Staubli VAL3: PlasticMain.pjx

--- PlasticMain.pjx ---
Parameters version=s7.0 stackSize=400000 millimeterUnit=true
Program file=__ts_english.pgx
Program file=__ts_german.pgx
Program file=__ts_swedish.pgx
Program file=_globals.pgx
Program file=changeLog.pgx
Program file=checkRobotPos.pgx
Program file=checkTaskStates.pgx
Program file=cleanUpDataBase.pgx
Program file=controlTasks.pgx
Program file=createLicense.pgx
Program file=detailedStack.pgx
Program file=loadApplication.pgx
Program file=loadLibraries.pgx
Program file=loadSysData.pgx
Program file=loadUserProgram.pgx
Program file=loadVersionInfo.pgx
Program file=logo.pgx
Program file=parseStackInfo.pgx
Program file=processEvents.pgx
Program file=run.pgx
Program file=saveApplication.pgx
Program file=start.pgx
Program file=startUpTask.pgx
Program file=status.pgx
Program file=stop.pgx
Program file=taskKill.pgx
Program file=taskKiller.pgx
Data file=PlasticMain.dtx
Library alias=rob path=Disk://Plastic/Prototypes/modRobot/modRobot.pjx autoload=false
Library alias=data path=Disk://Plastic/templates/sysDataTemplate/sysDataTemplate.pjx autoload=false
Library alias=secu path=Disk://Plastic/Prototypes/modSafety/modSafety.pjx autoload=false
Library alias=util path=Disk://Plastic/Prototypes/modBackup/modBackup.pjx autoload=false
Library alias=FUN path=Disk://Plastic/templates/tempSysFuncCall/tempSysFuncCall.pjx autoload=false
Library alias=fun path=Disk://Plastic/Prototypes/modFunction/modFunction.pjx autoload=false
Library alias=ui path=Disk://Plastic/Prototypes/modUserDisp/modUserDisp.pjx autoload=false
Library alias=prg path=Disk://Plastic/templates/tempUserProgram/tempUserProgram.pjx autoload=false
Library alias=USER path=Disk://Plastic/templates/tempIoUser/tempIoUser.pjx autoload=false
Library alias=app path=Disk://Plastic/templates/tempApplication/tempApplication.pjx
Library alias=appTmp path=Disk://Plastic/templates/tempApplication/tempApplication.pjx
Library alias=evt path=Disk://Plastic/Prototypes/modEvents/modEvents.pjx autoload=false
Library alias=SYS path=Disk://io_System/io_System.pjx
Library alias=str path=Disk://Libraries/stringHandling/stringHandling.pjx
Library alias=list path=Disk://Libraries/listHandling/listHandling.pjx
Library alias=upd path=Disk://Plastic/Prototypes/modUpdater/modUpdater.pjx autoload=false
Library alias=stat path=Disk://Plastic/Prototypes/modStatus/modStatus.pjx autoload=false
Library alias=lang path=Disk://Plastic/i18n/i18n.pjx
Library alias=db path=Disk://Plastic/Prototypes/modDatabase/modDatabase.pjx autoload=false
Library alias=usr path=Disk://Plastic/Prototypes/modUserIO/modUserIO.pjx autoload=false
Library alias=hw path=Disk://Libraries/hardware/hardware.pjx
Library alias=msl path=Disk://Plastic/Prototypes/modMsl/modMsl.pjx autoload=false
Library alias=customModule path=Disk://Plastic/Prototypes/modCustom/modCustom.pjx autoload=false
Library alias=userIO path=Disk://zUserIODef/zUserIODef.pjx autoload=false
Library alias=monitor path=Disk://Plastic/Prototypes/modMonitor/modMonitor.pjx autoload=false
Library alias=debug path=Disk://Libraries/debug/debug.pjx

--- PlasticMain.dtx ---
num nPLCRestartCnt
string programList
string sTaskName[3]
  [0] = "PLC_Main"
  [1] = "MP_MainPRG"
  [2] = "SR_HomeReturn"
string sVersion
string sBuildNumber
bool bFirstLoad = true
bool bStartUp
bool homeFlag
bool overrun
string sRawList
string sCopyRight = "Plastics (C) 2006-2011 V"

--- __ts_german.pgx ---
program __ts_german()
begin
  //
end

--- __ts_swedish.pgx ---
program __ts_swedish()
begin
  //
end

--- _globals.pgx ---
program _globals()
begin
    //\brief
  //
  //\version
  //4.3c
  //
//!version 4.3c
end

--- controlTasks.pgx ---
program controlTasks()
  local bool bResult
  local num nResult
begin
    //
  //\var bResult
  //\var nResult
  //
//=========================================================================
  // START PLC
  //=========================================================================
  if (taskStatus(sTaskName[0])==-1)
    taskCreate (sTaskName[0]),10,app:PLC_MainPLC()
  endIf
  // if PLC task is stopped due to an runtime error it should be restarted immediately
  if (taskStatus(sTaskName[0])>1) and nPLCRestartCnt<5
    if nPLCRestartCnt<5
      call ui:error("PLC task "+sTaskName[0]+" of "+data:sApplication+" died unexpectedly with error #"+toString(".0",taskStatus(sTaskName[0])))
      nPLCRestartCnt=nPLCRestartCnt+1
      nResult=1
    else
      call ui:question("PLC task "+sTaskName[0]+" died to often! Do you want to continue?",nResult)
      if nResult==1
        nPLCRestartCnt=0
      endIf
    endIf
    if nResult==1
      taskKill(sTaskName[0])
      delay(1)
      taskCreate (sTaskName[0]),10,app:PLC_MainPLC()
    endIf
  endIf
  //!change: 11.03.08, vdg: try to restart PLC task when robot leaves home position
  if !SYS:bRobotHome and homeFlag and nPLCRestartCnt>=5
    nPLCRestartCnt=0
  endIf
  homeFlag=SYS:bRobotHome
  //=========================================================================
  // START PRODUCTION CYCLE
  //=========================================================================
  if SYS:bStartProdCycle and SYS:bRobotHome and (taskStatus(sTaskName[1])==-1)
    SYS:bStartProdCycle=false
    call taskKill(sTaskName[2],bResult)
    if !bResult
      // killing the task failed, because it is being debugged?!
      call ui:popUp((("Cycle start not possible!/nPlease check if task HR_HomeReturn exists in task manager!")),0,false)
    else
      // inform operator that force recording is active
      if SYS:bRecordForce
        call ui:popUp((("Recording is active!/nDeactivate it in Advanced Settings->Test Run->Edit System Settings")),data:nMsgTimeOut,false)
      endIf
      resetMotion()
      restartMove()
      // reduce monitor speed to data:nSpeedAfterLoad if this is the first start cycle
      if SYS:bFirstRunAfterL
        ///TODO
        //$setSpeed(min(data:nSpeedAfterLoad,speedScale()))
        call fun:setSpeed(min(data:nSpeedAfterLoad,getMonitorSpeed()))
        // give the system some time to adjust the monitor speed before
        // MP_MainProgram is actually started
        delay(0.4)
        SYS:bFirstRunAfterL=false
        //
        //!change 18.05.06, vdg: activate test run after application has been loaded
        if data:setAutoTestRun
          data:setTestRun=true
        endIf
      endIf
      //!change 22.08.06, vdg: reset area test
      call secu:primeAreaTest()
      logMsg("Production started")
      // disallow to start IMM if end cycle is active
      SYS:bStartInEndCycl=false
      // allow to cancel end cycle function by operator
      SYS:bCancelEndCycle=true
      //!Issue 22: call user event program
      call prg:onAppStart()
      taskCreate (sTaskName[1]),10,app:MP_MainProgram()
      SYS:bTotalHome=false
    endIf
  endIf
  // reset state if main task has ended
  if taskStatus(sTaskName[1])==-1 and SYS:nStateRobot>=10 and SYS:nStateRobot<26
    SYS:nStateRobot=0
  endIf
  //!change 12.07.06, vdg: reset automatic timer if robot cycle is not running or
  // robot power is disabled or working mode is not automatic
  if (taskStatus(sTaskName[1])!=1) or !isPowered() or (workingMode()<3)
    call ui:resetAutoTimer()
  endIf
  //=========================================================================
  // START HOME RETURN CYCLE
  //=========================================================================
  if SYS:bStartHomeCycle and (taskStatus(sTaskName[2])==-1)
    logMsg("Production stopped")
    //!issue 48: home return not possible if main task is being debugged
    // This is a work around for a Val3 bug which makes the
    // program block in taskKill() when the task is currently being debugged
    //taskKill(sTaskName[1])
    // try to kill the task
    call taskKill(sTaskName[1],bResult)
    if !bResult
      // killing the task failed, because it is being debugged?!
      call ui:popUp("Home return not possible!/nPlease verify that task MP_MainPrg is not debuuged in task manager",0,false)
      // reset state machine robMotionCtrl
      SYS:nStateRobot=0
    else
      if SYS:bTotalHome
        //!issue 22
        if data:setResetPLCOnHo
          call prg:resetPLC()
        endIf
      endIf
      //!change 08.06.06, vdg: wait until task is killed by system
      wait(taskStatus(sTaskName[1])==-1)
      //!Issue 22: call user event program
      call prg:onAppStop()
      //!issue 48
      // go to next step in state machine robMotionCtrl
      SYS:nStateRobot=32
      resetMotion()
      restartMove()
      taskCreate (sTaskName[2]),10,app:HR_HomeReturn()
      //!Issue 22: call user event program
      call prg:onHomeStart(SYS:bTotalHome)
    endIf
    SYS:bStartHomeCycle=false
  endIf
  //=========================================================================
  // CANCEL HOME RETURN CYCLE
  //=========================================================================
  //!fix vdg, 13.03.08: Reset SYS:bCancelHomeCycl event if home return is not active
  if SYS:bCancelHomeCycl
    if (taskStatus(sTaskName[2])!=-1)
      stopMove()
      call taskKill(sTaskName[2],bResult)
      if !bResult
        // killing the task failed, because it is being debugged?!
        call ui:popUp("Cycle start not possible!/nPlease verify that task HR_HomeReturn is not debugged in task manager!",0,false)
      else
        resetMotion()
        SYS:bCancelHomeCycl=false
      endIf
    else
      SYS:bCancelHomeCycl=false
    endIf
  endIf
end

--- createLicense.pgx ---
program createLicense()
  local string txt[6]
  local string orderNumber
  local num i
 begin
    //\brief
  // Create a license key for the robot system. License key information is saved
  // in system data library
  //
  //\var txt
  //\var orderNumber
  //\var i
  //
//!brief
  // Create a license key for the robot system. License key information is saved
  // in system data library
  //
  orderNumber=getVersion("serialNumber")
  txt=""
  //!issue 36
  if data:libLoad("zData")==0
    call list:resizeNum(data:nLic,len(orderNumber))
    data:sMachineNumber=orderNumber
    for i=0 to size(data:nLic)-1
      data:nLic[i]=asc(orderNumber,i)*(i+1)
      txt=txt+toString("",asc(orderNumber,i)*(i+1))+", "
    endFor
    call data:saveData()
    popUpMsg(txt)
  else
    popUpMsg("Loading the data library failed!")
  endIf
end

--- detailedStack.pgx ---
program detailedStack()
  local num i
  local num nTaskStatus
  local num count
  local num j
  local string stack[20]
begin
    //\brief
  //Write detailed stack info to log
  //\var i
  //\var nTaskStatus
  //\var count
  //\var j
  //\var stack
  //
//!brief
  //Write detailed stack info to log
  for i=0 to size(sTaskName)-1
    logMsg("Stack Information for task: "+sTaskName[i])
    nTaskStatus=taskStatus(sTaskName[i])
    // suspend the task
    if nTaskStatus==1
      taskSuspend(sTaskName[i])
    endIf
    // wait until task stopped
    wait(taskStatus(sTaskName[i])!=1)
    // retrieve call stack
    count=$taskCallStack(sTaskName[i],stack)
    // write call stack to log
    for j=0 to count-1
      logMsg(stack[j])
    endFor
    // resume task if it was active when entering this routine
    if nTaskStatus==1
      taskResume(sTaskName[i],0)
    endIf
  endFor
end

--- loadSysData.pgx ---
program loadSysData(bool& bResult_[], bool& bSetupLicense_[])
  local num nResult
begin
    //
  //\var nResult
  //\param bResult_
  //\param bSetupLicense_
  //
put("Loading Data for: "+libPath()+" :")
  nResult=data:libLoad("zData")
  bSetupLicense_=false
  //
  switch true
    // library loaded
    case nResult==0
      putln("ok")

    break
    // zData library does not exist yet, so we save the template
    // as zData
    case nResult>=30
      bResult_=false
      logMsg("zData not found!")
      // reload template
      nResult=data:libLoad("Plastic/templates/sysDataTemplate")
      if nResult==0
        // save template as zData
        nResult=data:libSave("zData")
        if nResult==0
          logMsg("zData recreated from template")
          bResult_=true
          // if profile 'swiss-system' is active also force creation of license
          if getProfile()=="swiss-system"
            bSetupLicense_=true
          else
            popUpMsg("A new zData library has been created. Please reinstall runtime license!")
          endIf
        else
          logMsg("Creating zData failed!")
        endIf
      endIf
    break
    // library load failed for some other reason
    default
      putln("failed")
      putln("Checking data dependencies")
      call upd:checkDepend()
      bResult_=false
    break
  endSwitch
end

--- parseStackInfo.pgx ---
program parseStackInfo(string stackInfo_, string& library_[], string& program_[], num& line_[], string& code_[])
  local bool error
  local string dummy
begin
    //
  //\var error
  //\var dummy
  //\param stackInfo_
  //\param library_
  //\param program_
  //\param line_
  //\param code_
  //
if len(stackInfo_)>0
    library_=left(stackInfo_,find(stackInfo_,":"))
    stackInfo_=right(stackInfo_,len(stackInfo_)-find(stackInfo_,":")-1)
    program_=left(stackInfo_,find(stackInfo_,")")+1)
    stackInfo_=right(stackInfo_,len(stackInfo_)-find(stackInfo_,")")-1)
    stackInfo_=right(stackInfo_,len(stackInfo_)-find(stackInfo_,"ne")-3)
    dummy=stackInfo_
    dummy=toNum(dummy,line_,error)
    stackInfo_=right(stackInfo_,len(stackInfo_)-find(stackInfo_,":")-1)
    code_=stackInfo_
  endIf
end

--- processEvents.pgx ---
program processEvents()
  local num event
  local num idx
  local num nResult
  local num char
begin
    //
  //\var event
  //\var idx
  //\var nResult
  //\var char
  //
// check pending events
  call evt:getEvent(event)
  switch event
    // application load event
    case evt:evtLoadApp
      // clear any non persistent status messages
      call stat:clearStatusMsg(false)
      // Aquire stat:mutex in order to avoid calls to the status list control
      // (stat:addStatusMsg(), etc) when the user application task are being called.
      // This should avoid a race condition which was first observed in Hammarplast application.
      call stat:aquireMutex()
      // stop application tasks
      taskKill(sTaskName[0])
      taskKill(sTaskName[1])
      taskKill(sTaskName[2])
      //!change 05.07.06, vdg: wait until all tasks are killed
      for idx=0 to size(sTaskName)-1
        wait(taskStatus(sTaskName[idx])==-1)
      endFor
      call stat:releaseMutex()
      resetMotion()
      disablePower()
      call loadApplication(evt:sEventParam[0])
      //!TODO
      if bFirstLoad
        //call loadApplication(evt:sEventParam[0])
        bFirstLoad=false
      endIf
      // do a total home return after loading the new application
      SYS:bTotalHome=true
      // inform ui that event has been processed
      call evt:resetEvent()
    break
    // save application event
    case evt:evtSaveApp
      call saveApplication()
      // inform ui that event has been processed
      call evt:resetEvent()
    break
    case evt:evtRunWizard
      //call wiz:wzNewApp()
      call evt:resetEvent()
    break
    case evt:evtBackup
      call util:backup(evt:sEventParam[0],nResult)
      call evt:resetEvent()
    break
    case evt:evtUpdStatusTxt
      call stat:update()
      call evt:resetEvent()
    break
    case evt:evtStackInfo
      call detailedStack()
      call evt:resetEvent()
    break
    //  if sioGet(io:slave,char)==1
    //    char=io:slave
    //    if true
    //      call stat:sendStatus(io:slave)
    //      clearBuffer(io:slave)
    //    endIf
    //  endIf
  endSwitch
end

--- status.pgx ---
program status()
  local num count
  local string callStack
  local string library
  local string program
  local num line
  local string code
begin
    //
  //\var count
  //\var callStack
  //\var library
  //\var program
  //\var line
  //\var code
  //
while true
    count=$taskCallStack(sTaskName[1],callStack)
    call parseStackInfo(callStack,library,program,line,code)
    if program=="SP_Traj"
      call list:resizeString(programList,max(size(programList),line))
      programList[line]=code
    endIf
  endWhile
end

--- taskKill.pgx ---
program taskKill(string sTaskName_, bool& bResult_[])
  local num idx
begin
    //\brief
  //The program tries to kill task sTaskName_. bResult_ is false if it does not
  // succeed within 2 sec
  //\var idx
  //\param sTaskName_ The name of the task that should be killed
  //\param bResult_ The result of the kill operation
  //
  // find free task
  //
//!brief
  //The program tries to kill task sTaskName_. bResult_ is false if it does not
  // succeed within 2 sec
  //!param sTaskName_ : The name of the task that should be killed
  //!param bResult_   : The result of the kill operation
  //
  // find free task
  idx=0
  while taskStatus("killer"+toString("",idx))!=-1
    idx=idx+1
  endWhile
  taskCreate "killer"+toString("",idx),1,taskKiller(sTaskName_)
  if !watch(taskStatus("killer"+toString("",idx))==-1,2)
    bResult_=false
    taskKill("killer"+toString("",idx))
  else
    bResult_=true
  endIf
end

--- taskKiller.pgx ---
program taskKiller(string sTask_)
begin
    //
  //\param sTask_
  //
taskKill(sTask_)
end
